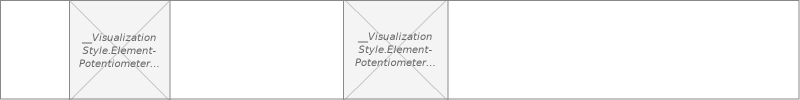
VISUALIZATION Nav  // 800x100
    Image (343,-2 105x103)
    Image (69,0 101x101)
        OnMouseDown: change screen: Safty_Zones_and_Modes
END_VISUALIZATION

(* stored: Version 1.1.0.1, ProductVersion 3.1.4024.12
   Visu Nav: Id {62736221-5416-4347-a636-1b4a4d544294} *)
